(* IEC 61131-3 sources: Industry-PLC-LLM/data/PLCBEAD_repo/PLCBEAD_PLCEmbed-main/PLC-BEAD/Source/GEB/M_T, 1 file *)

(* ---- M_T.ST ---- *)
FUNCTION_BLOCK T_PLC_MS_block
	VAR_OUTPUT
		T_PLC_MS :	UDINT;
	END_VAR

	VAR
		PLC_TICKS_PER_SEC :	INT;
		PLC_SYS_TICK_CNT :	DINT;
	END_VAR

	VAR
		debug :	BOOL;(*Debug-Mode ON / OFF*)
		N :	INT;(*Debug-Faktor*)
		Offset :	UDINT;(*Debug-Offset*)
		temp :	DWORD := DWORD#1;(*Debug-Offset*)
		MODE :	BOOL;(*modus*)
		faktor :	UDINT;(*Systemtakt-Faktor*)
		init :	BOOL;
		v_plc_ticks_per_sec :	UDINT;
		base :	UDINT := UDINT#1000;
	END_VAR

	IF init = FALSE THEN
		v_plc_ticks_per_sec := INT_TO_UDINT(PLC_TICKS_PER_SEC);
		IF v_plc_ticks_per_sec = UDINT#1024 THEN
			faktor := UDINT#1;
			MODE := FALSE;
		ELSIF v_plc_ticks_per_sec > UDINT#0 THEN
			IF v_plc_ticks_per_sec <= base THEN
				faktor := base / v_plc_ticks_per_sec;
				MODE := FALSE;
			ELSE
				faktor := v_plc_ticks_per_sec / base;
				MODE := TRUE;
			END_IF;
		ELSE
			faktor := UDINT#1;
		END_IF;
		init := TRUE;
	END_IF;

	IF MODE THEN
		T_PLC_MS := DINT_TO_UDINT(PLC_SYS_TICK_CNT) / faktor;
	ELSE
		T_PLC_MS := DINT_TO_UDINT(PLC_SYS_TICK_CNT) * faktor;
	END_IF;

	IF debug THEN
		T_PLC_MS := (DWORD_TO_UDINT(SHL(UDINT_TO_DWORD(T_PLC_MS),N) OR SHL(temp,N)) - UDINT#1) + Offset;
	END_IF;
END_FUNCTION_BLOCK

FUNCTION_BLOCK M_T_Block

	VAR_INPUT
		IN :	BOOL;
		TMAX :	TIME := t#10d;
		RST :	BOOL;
	END_VAR

	VAR_OUTPUT
		PT :	TIME;
		ET :	TIME;
	END_VAR

	VAR
		edge :	BOOL;
		START :	TIME;
		TX :	TIME;
		T_PLC_MS :	T_PLC_MS_block;
	END_VAR

	(*@KEY@: WORKSHEET
	NAME: M_T
	IEC_LANGUAGE: ST
	*)
	(* read system timer *)
	T_PLC_MS();
	TX:= UDINT_TO_TIME(T_PLC_MS.T_PLC_MS);

	IF RST OR ET >= TMAX THEN
		PT := t#0s;
		ET := PT;
	ELSIF IN THEN
		IF NOT edge THEN START := TX; END_IF;
		ET := SUB_TIME(TX, START);
	ELSE
		PT := ET;
	END_IF;
	edge := IN;

END_FUNCTION_BLOCK

PROGRAM program0

	VAR
		IN :	BOOL;
		TMAX :	TIME := t#10d;
		RST :	BOOL;

		PT :	TIME;
		ET :	TIME;

		func_block : M_T_Block;
	END_VAR
	func_block.IN := IN;
	func_block.TMAX := TMAX;
	func_block.RST := RST;

	func_block();
	PT := func_block.PT;
	ET := func_block.ET;

END_PROGRAM
